# EPICS autosave request: iocs/uvcIOC/iocBoot/iocADUVC/auto_settings.req
file "ADUVC_settings.req",          P=$(P),  R=cam1:
file "NDStdArrays_settings.req",    P=$(P),  R=image1:
file "commonPlugin_settings.req",   P=$(P)
